{attribute 'qualified_only'}
{attribute 'strict'}
TYPE DeleteFilesState :
(
	Idle := 0,
  SearchNextFile,
  WaitUntilExecutionDone,
  ProcessFoundFiles,
  CheckIfFileIsDirectory,
  CheckFileTime,
  DeleteFile,
  FileDeleted
);
END_TYPE

(* stored: Version 1.1.0.1
   DUT DeleteFilesState: Id {01a80c6b-14dd-4079-8b88-25b2a5d0c1d3} *)
